Yaskawa INFORM job: X4_NOWY_SPR.JBI

/JOB
//NAME X4_NOWY_SPR
//POS
///NPOS 55,55,55,4,0,0
///TOOL 0
///POSTYPE PULSE
///PULSE
C00000=3270,-119374,-120744,-349,28960,82703
C00001=-89062,-116132,-100192,-547,17977,82798
C00002=-131984,-112240,-101963,23516,27648,71601
C00003=-137270,-105655,-98262,29917,28765,68085
C00004=-137697,-85179,-88546,26822,32933,69721
C00005=-137697,-85186,-87960,27077,32607,69586
C00006=-137697,-85179,-88546,26822,32933,69721
C00007=-144714,-132270,-106347,49581,25358,58340
C00008=-143520,-63582,-101695,13975,78864,74898
C00009=-143548,-56359,-97531,13944,79985,75017
C00010=-142914,-51821,-94992,13604,80642,75280
C00011=-143548,-56359,-97531,13944,79985,75017
C00012=-147878,-88611,-112493,16486,73583,72842
C00013=-102037,-133341,-129837,2447,31472,80379
C00014=-106484,-83959,-106846,6584,39726,78275
C00015=-107145,-76189,-102742,7107,41235,78086
C00016=-107145,-76638,-102287,7180,40729,78043
C00017=-107145,-76189,-102742,7107,41235,78086
C00018=-104118,-111508,-118221,4675,32446,79000
C00019=-94830,-22842,-101591,1863,98627,85949
C00020=-96751,-14552,-95564,2851,99211,85552
C00021=-97220,-11825,-93542,3094,99378,85457
C00022=-96751,-14552,-95564,2851,99211,85552
C00023=-90289,-50383,-117683,-451,94353,86933
C00024=-113680,-103951,-120589,13317,46690,76070
C00025=-117692,-43924,-75065,61492,51873,58717
C00026=-118714,-28685,-66281,64145,60532,60129
C00027=-113945,-28124,-65864,61617,57807,60938
C00028=-114902,-26070,-64609,63051,59070,60714
C00029=-127850,-26661,-63451,72108,65262,58732
C00030=-130557,-33924,-68329,73549,66718,58095
C00031=-106572,-58848,-93942,15426,45804,80121
C00032=-106805,-57460,-92531,15692,45693,80004
C00033=-102131,-55289,-91366,11012,45402,81938
C00034=-108857,-71296,-101220,18205,44385,78853
C00035=-110435,-82200,-106133,1038,40006,86002
C00036=-110257,-62003,-97964,607,48269,86053
C00037=-105614,-60279,-97081,-3756,48691,87855
C00038=-103782,-78639,-107364,-5746,45692,88747
C00039=-132684,-130914,-127982,52253,49571,61610
C00040=-139278,-129792,-110794,83567,32161,45718
C00041=-120590,-62989,-101418,16330,54617,61245
C00042=-125724,-56772,-97284,25246,57738,57639
C00043=-122888,-57846,-96478,25783,55309,59395
C00044=-127522,-66713,-102028,29694,55636,57651
C00045=-107332,-64864,-101121,-24429,54104,80168
C00046=-108124,-58631,-96750,-23652,54375,79793
C00047=-114127,-60353,-97642,-18825,52712,77837
C00048=-113976,-63835,-99856,-19057,52338,77968
C00049=-99038,-37275,-75810,-62036,67050,86790
C00050=-101956,-36523,-73710,-63796,66102,86763
C00051=-95054,-53921,-86066,-55693,56200,84395
C00052=-78339,-85415,-97950,-74258,61103,88238
C00053=-70048,-95947,-100914,-80606,65818,89400
C00054=3270,-119374,-120744,-349,28960,82703
BC00000=132383,666204,620608
BC00001=246848,666204,238820
BC00002=314536,666204,238819
BC00003=314494,666205,238814
BC00004=314494,666205,238814
BC00005=314494,666205,238814
BC00006=314494,666205,238814
BC00007=314494,666205,238814
BC00008=314494,666205,238814
BC00009=314494,666205,238814
BC00010=314494,666205,238814
BC00011=314494,666205,238814
BC00012=314494,666205,238814
BC00013=89204,663597,111569
BC00014=89204,663597,111569
BC00015=89204,663597,111569
BC00016=89204,663597,111569
BC00017=89204,663597,111569
BC00018=89204,663597,111569
BC00019=89204,663597,111569
BC00020=89204,663597,111569
BC00021=89204,663597,111569
BC00022=89204,663597,111569
BC00023=89204,663597,111569
BC00024=89204,663597,111569
BC00025=89204,663597,111569
BC00026=89204,663597,111569
BC00027=89204,663597,111569
BC00028=89204,663597,111569
BC00029=89204,663597,111569
BC00030=89204,663597,111569
BC00031=89204,663597,111569
BC00032=89204,663597,111569
BC00033=89204,663597,111569
BC00034=89204,663597,111569
BC00035=89204,663597,111569
BC00036=89204,663597,111569
BC00037=89204,663597,111569
BC00038=89204,663597,111569
BC00039=89204,665553,111569
BC00040=294804,665553,111569
BC00041=294804,665553,111569
BC00042=294804,665553,111569
BC00043=294804,665553,111569
BC00044=294804,665553,111569
BC00045=294804,665553,111569
BC00046=294804,665553,111569
BC00047=294804,665553,111569
BC00048=294804,665553,111569
BC00049=294804,665553,111569
BC00050=294804,665553,111567
BC00051=294804,665553,111567
BC00052=294804,665553,111567
BC00053=294804,665553,111567
BC00054=132383,666204,620608
EC00000=-77843,-555115
EC00001=-77843,-555115
EC00002=-77843,-555115
EC00003=-77844,-555114
EC00004=-77844,-555114
EC00005=-77844,-555114
EC00006=-77844,-555114
EC00007=-77844,-555114
EC00008=-77844,-555114
EC00009=-77844,-555114
EC00010=-77844,-555114
EC00011=-77844,-555114
EC00012=-77844,-555114
EC00013=-77844,-555116
EC00014=-77844,-555116
EC00015=-77844,-555116
EC00016=-77844,-555116
EC00017=-77844,-555116
EC00018=-77844,-555116
EC00019=-77844,-555116
EC00020=-77844,-555116
EC00021=-77844,-555116
EC00022=-77844,-555116
EC00023=-77844,-555116
EC00024=-77844,-555116
EC00025=-77844,-555116
EC00026=-77844,-555116
EC00027=-77844,-555116
EC00028=-77844,-555116
EC00029=-77844,-555116
EC00030=-77844,-555116
EC00031=-77844,-555116
EC00032=-77844,-555116
EC00033=-77844,-555116
EC00034=-77844,-555116
EC00035=-77844,-555116
EC00036=-77844,-555116
EC00037=-77844,-555116
EC00038=-77844,-555116
EC00039=-77844,-555116
EC00040=-77844,-555116
EC00041=-77844,-555116
EC00042=-77844,-555116
EC00043=-77844,-555116
EC00044=-77844,-555116
EC00045=-77844,-555116
EC00046=-77844,-555116
EC00047=-77844,-555116
EC00048=-77844,-555116
EC00049=-77844,-555116
EC00050=-77844,-555116
EC00051=-77844,-555116
EC00052=-77844,-555116
EC00053=-77844,-555116
EC00054=-77843,-555115
///POSTYPE BASE
///RECTAN
///RCONF 0,0,0,0,0,0,0,0,0,0,0,0,0,0,0,0,0,0,0,0,0,0,0,0
P00006=0.222,-3.123,-1.508,0.0000,0.0000,0.0000
P00031=1.853,-0.001,-1.549,0.0000,0.0000,0.0000
P00032=1.957,0.503,-7.217,0.0000,0.0000,0.0000
///RCONF 0,0,0,0,1,0,0,0,0,0,0,0,0,0,0,0,0,0,0,0,0,0,0,0
P00033=-0.123,0.612,-5.012,0.0000,0.0000,0.0000
//INST
///DATE 2024/04/03 18:52
///COMM BRAKUJACE SPOINY
///ATTR SC,RW
///GROUP1 RB1,BS1
///GROUP2 ST1
NOP
MOVJ C00000 BC00000 VJ=100.00  +MOVJ EC00000 VJ=100.00
MOVJ C00001 BC00001 VJ=100.00  +MOVJ EC00001 VJ=100.00
MOVJ C00002 BC00002 VJ=40.00  +MOVJ EC00002 VJ=100.00
SMOVL C00003 BC00003 V=150.0  +MOVJ EC00003
SMOVL C00004 BC00004 V=100.0  +MOVJ EC00004
SREFP 3 C00005 BC00005  +REFP EC00005
CALL JOB:SEARCH-R1-S13D
SET P031 P006
SFTON3D P031
SMOVL C00006 BC00006 V=100.0  +MOVJ EC00006
SMOVL C00007 BC00007 V=333.3  +MOVJ EC00007
SMOVL C00008 BC00008 V=333.3  +MOVJ EC00008
SMOVL C00009 BC00009 V=333.3  +MOVJ EC00009
SREFP 3 C00010 BC00010  +REFP EC00010
CALL JOB:SEARCH-R1-S13D
SET P031 P006
SFTON3D P031
SMOVL C00011 BC00011 V=150.0  +MOVJ EC00011
SFTOF3D
SMOVL C00012 BC00012 V=500.0  +MOVJ EC00012
SMOVL C00013 BC00013 V=666.7  +MOVJ EC00013
SMOVL C00014 BC00014 V=333.3  +MOVJ EC00014
SMOVL C00015 BC00015 V=100.0  +MOVJ EC00015
SREFP 3 C00016 BC00016  +REFP EC00016
CALL JOB:SEARCH-R1-S13D
SET P033 P006
SFTON3D P033
SMOVL C00017 BC00017 V=100.0  +MOVJ EC00017
SMOVL C00018 BC00018 V=500.0  +MOVJ EC00018
SMOVL C00019 BC00019 V=500.0  +MOVJ EC00019
SMOVL C00020 BC00020 V=166.7  +MOVJ EC00020
SREFP 3 C00021 BC00021  +REFP EC00021
CALL JOB:SEARCH-R1-S13D
SET P033 P006
SFTON3D P033
SMOVL C00022 BC00022 V=100.0  +MOVJ EC00022
SFTOF3D
SMOVL C00023 BC00023 V=333.3  +MOVJ EC00023
SMOVL C00024 BC00024 V=333.3  +MOVJ EC00024
SMOVL C00025 BC00025 V=150.0  +MOVJ EC00025
MACRO1 MJ#(0) ARGF14
SMOVL C00026 BC00026 V=333.3  +MOVJ EC00026
ARCON
SMOVL C00027 BC00027 V=10.0  +MOVJ EC00027
ARCOF
SMOVL C00028 BC00028 V=166.7  +MOVJ EC00028
SMOVL C00029 BC00029 V=166.7  +MOVJ EC00029
SMOVL C00030 BC00030 V=166.7  +MOVJ EC00030
SMOVL C00031 BC00031 V=166.7  +MOVJ EC00031
SMOVL C00032 BC00032 V=166.7  +MOVJ EC00032
ARCON
SMOVL C00033 BC00033 V=10.0  +MOVJ EC00033
ARCOF
SMOVL C00034 BC00034 V=166.7  +MOVJ EC00034
SFTOF3D
SMOVL C00035 BC00035 V=166.7  +MOVJ EC00035
SFTON3D P033
SMOVL C00036 BC00036 V=166.7  +MOVJ EC00036
ARCON
SMOVL C00037 BC00037 V=10.0  +MOVJ EC00037
ARCOF
SMOVL C00038 BC00038 V=250.0  +MOVJ EC00038
SFTOF3D
SMOVL C00039 BC00039 V=666.7  +MOVJ EC00039
SMOVL C00040 BC00040 V=666.7  +MOVJ EC00040
SMOVL C00041 BC00041 V=333.3  +MOVJ EC00041
SFTON3D P031
SMOVL C00042 BC00042 V=166.7  +MOVJ EC00042
ARCON
SMOVL C00043 BC00043 V=10.0  +MOVJ EC00043
ARCOF
SMOVL C00044 BC00044 V=166.7  +MOVJ EC00044
SMOVL C00045 BC00045 V=166.7  +MOVJ EC00045
SFTON3D P032
SMOVL C00046 BC00046 V=166.7  +MOVJ EC00046
ARCON
SMOVL C00047 BC00047 V=10.0  +MOVJ EC00047
ARCOF
SMOVL C00048 BC00048 V=133.3  +MOVJ EC00048
SMOVL C00049 BC00049 V=250.0  +MOVJ EC00049
ARCON
SMOVL C00050 BC00050 V=10.0  +MOVJ EC00050
ARCOF
SMOVL C00051 BC00051 V=333.3  +MOVJ EC00051
SFTOF3D
SMOVL C00052 BC00052 V=666.7  +MOVJ EC00052
MOVJ C00053 BC00053 VJ=100.00  +MOVJ EC00053 VJ=100.00
MOVJ C00054 BC00054 VJ=100.00  +MOVJ EC00054 VJ=100.00
END
